(* PLC project mode, Dassault Systèmes ControlBuild 2024x *)
(* stored: creationDateTime 2023-10-03T11:13:44-01:00 *)

FUNCTION_BLOCK drill.mode
  VAR_INPUT
    powerUpPB : BOOL := false;
    startCyclePB : BOOL := false;
    emergencyStop : BOOL := false;
    batchCycle : BOOL := false;
    pieceCycle : BOOL := false;
    autoSwitch : BOOL := false;
    manualSwitch : BOOL := false;
  END_VAR
  VAR_INPUT
    cycleEnd : BOOL := false;
    acknowledgePB : BOOL := false;
  END_VAR
  VAR_OUTPUT
    live : BOOL := false;
  END_VAR
  VAR_OUTPUT
    autoMode : BOOL := false;
    manualMode : BOOL := false;
  END_VAR
  VAR_OUTPUT
    emptyProd : BOOL := false;
    unitProd : BOOL := false;
    batchProd : BOOL := false;
  END_VAR
  VAR
    emergencyState : BOOL := false;
  END_VAR
  VAR  (* added by the conversion: wires and edge detectors of the diagram *)
    R_TRIG1 : R_TRIG;
    F_TRIG2 : F_TRIG;
    R_TRIG3 : R_TRIG;
    F_TRIG4 : F_TRIG;
  END_VAR

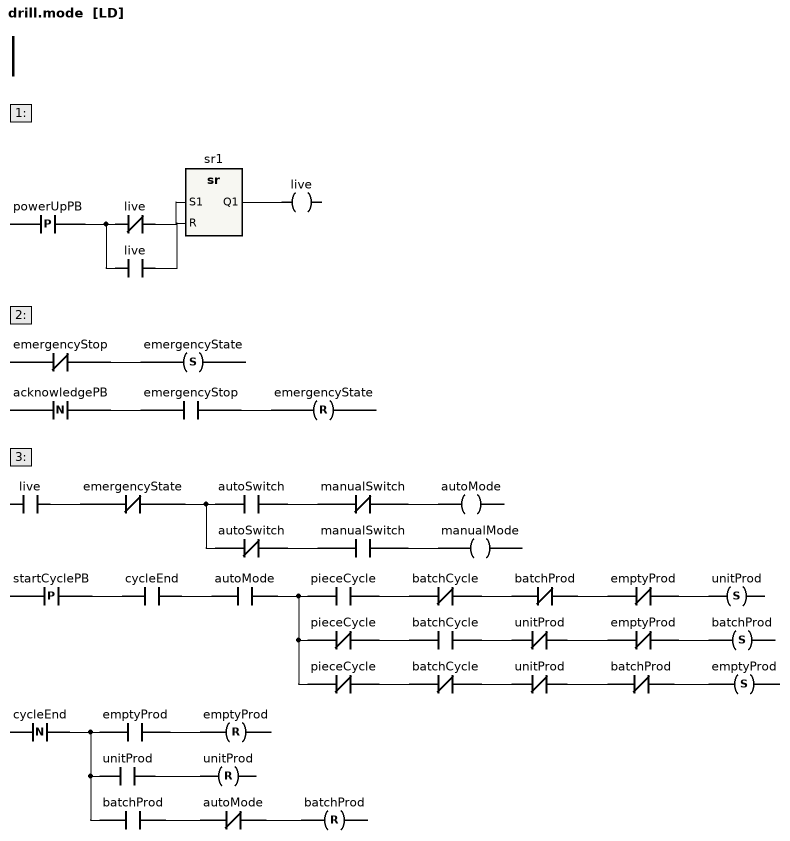
(* LD diagram, written out as Structured Text *)
1:
R_TRIG1(CLK := powerUpPB);
sr1(S1 := R_TRIG1.Q AND NOT live, R := R_TRIG1.Q AND live);
live := sr1.Q1;
2:
IF NOT emergencyStop THEN emergencyState := TRUE; END_IF;
F_TRIG2(CLK := acknowledgePB);
IF F_TRIG2.Q AND emergencyStop THEN emergencyState := FALSE; END_IF;
3:
autoMode := live AND NOT emergencyState AND autoSwitch AND NOT manualSwitch;
manualMode := live AND NOT emergencyState AND NOT autoSwitch AND manualSwitch;
R_TRIG3(CLK := startCyclePB);
IF R_TRIG3.Q AND cycleEnd AND autoMode AND pieceCycle AND NOT batchCycle AND NOT batchProd AND NOT emptyProd THEN unitProd := TRUE; END_IF;
IF R_TRIG3.Q AND cycleEnd AND autoMode AND NOT pieceCycle AND batchCycle AND NOT unitProd AND NOT emptyProd THEN batchProd := TRUE; END_IF;
IF R_TRIG3.Q AND cycleEnd AND autoMode AND NOT pieceCycle AND NOT batchCycle AND NOT unitProd AND NOT batchProd THEN emptyProd := TRUE; END_IF;
F_TRIG4(CLK := cycleEnd);
IF F_TRIG4.Q AND emptyProd THEN emptyProd := FALSE; END_IF;
IF F_TRIG4.Q AND unitProd THEN unitProd := FALSE; END_IF;
IF F_TRIG4.Q AND batchProd AND NOT autoMode THEN batchProd := FALSE; END_IF;
END_FUNCTION_BLOCK
